FUNCTION_BLOCK FB_MixedGuid
VAR
END_VAR

END_FUNCTION_BLOCK

(* stored: Version 1.1.0.1, ProductVersion 3.1.4024.12
   POU FB_MixedGuid: Id {A1B2C3D4-E5F6-7890-ABCD-EF1234567890}, SpecialFunc None *)
